FUNCTION_BLOCK FB_LinearGovernor
VAR_INPUT
	i_stCurrentBeamParams	:	ST_BeamParams; //Link to global beam params
	i_xMPSOverride			:	BOOL; //True releases MPS limits after a delay
	i_xTransitionRequested	:	BOOL; //Set true to request a transition
	i_xResetMPSFault	:	BOOL; //Set true to clear MPS fault 
END_VAR
VAR_OUTPUT
	q_xTransitionPermitted	:	BOOL; //True when governor has released restrictions
	q_xFault	:	BOOL; //Set if MC_Power has an error, or override mode is requested
END_VAR
VAR_IN_OUT
	stDevice	:	ST_Device; //The governed
	Arbiter	:	FB_Arbiter;
END_VAR
VAR
	mcPower	:	MC_Power;
	
	xActuatorPositiveEnable: BOOL;
	xActuatorNegativeEnable: BOOL;
	
	xMPSPositiveEnable	:	BOOL;
	xMPSNegativeEnable	:	BOOL;
	lrPosition: LREAL;
	
	lrLatchedTargetPosition	:	LREAL;
	lrLatchedTargetTolerance	:	LREAL;
	
	lrMPSUpperLimit: LREAL;
	lrMPSLowerLimit: LREAL;
	rtNewState: R_TRIG;
	xTransitionOK: BOOL;
	
	tonMPSOverrideMode	:	TON := (
		PT := T#5S
	);
	
	srMPSFault	:	SR;
	// Actuator out of bounds fault
	xActuatorOOB: BOOL;
	xBeamParametersSafe: BOOL;
END_VAR


lrPosition := stDevice.stAxis.NcToPlc.ActPos;

//MPS Faults
//Fault if the position is outside of the permitted range
//Allow for transitions
IF xTransitionOK THEN
	//Extend range to include target state
ELSE
	//Calculate the limit positions for MPS based on current state
	lrMPSUpperLimit := lrLatchedTargetPosition + lrLatchedTargetTolerance/2;
	lrMPSLowerLimit := lrLatchedTargetPosition - lrLatchedTargetTolerance/2;
END_IF

//Latch the MPS fault
srMPSFault.SET1 := xActuatorOOB;
srMPSFault(RESET:=i_xResetMPSFault); 

//MPS limit switch logic


//Evaluate MPS limit states
xMPSPositiveEnable := lrPosition <= lrMPSUpperLimit;
xMPSNegativeEnable := lrPosition >= lrMPSLowerLimit;

//Determine if the MPS limits can be lifted
IF i_xTransitionRequested THEN
	Arbiter.A_VerifyAssertion(
		i_nStateID := stDevice.stTransitionState.nStateRef
	);
	xTransitionOK := Arbiter.q_xStateIDFound;
ELSE
	xTransitionOK := FALSE;
END_IF

//MPS override
(* In override mode, the device will be free to move anywhere within it's travel range *)
//Permit motion after a small delay
tonMPSOverrideMode(IN:=i_xMPSOverride);

//Virtual limit switch evaluation
xActuatorPositiveEnable	:= stDevice.i_xHiLim AND lrPosition <= stDevice.lrUpperPositionLimit;
xActuatorNegativeEnable	:= stDevice.i_xLoLim AND lrPosition <= stDevice.lrLowerPositionLimit;

//Final Limit switch evaluation
mcPower.Enable_Positive := xActuatorPositiveEnable AND (tonMPSOverrideMode.Q OR xMPSPositiveEnable);
mcPower.Enable_Negative := xActuatorNegativeEnable AND (tonMPSOverrideMode.Q OR xMPSNegativeEnable);

mcPower(
	Axis := stDevice.stAxis,
	Enable := stDevice.xEnable //link to device enable <TODO>
);

//An mcPower error or MPS override, or MPS fault, produces a fault. Faults can be masked by veto devices.
q_xFault := mcPower.Error OR i_xMPSOverride OR srMPSFault.Q1;

END_FUNCTION_BLOCK

(* stored: Version 1.1.0.1, ProductVersion 3.1.4022.12
   POU FB_LinearGovernor: Id {ef40f951-1e56-0d26-34ec-87da9b08d3b7}, SpecialFunc None *)
